% RSLogix 500 project Project 4.RSS, saved by version 8.30.00.16 %
PROJECT "UNTITLED"    % processor: Bul.1763 MicroLogix 1100 Series B %

PROGRAM FILES
  LAD 2 "MAIN"  5 rungs
  LAD 3 "IO"  8 rungs
  LAD 4 "CYCLE"  6 rungs
  LAD 5 "CONTROLS"  11 rungs

DATA FILES
  O0 OUTPUT  4 elements
  I1 INPUT  6 elements
  S2 STATUS  66 elements
  B3 BINARY  1 elements
  T4 TIMER  3 elements
  C5 COUNTER  1 elements
  R6 CONTROL  1 elements
  N7 INTEGER  3 elements
  F8 FLOAT  1 elements

LADDER 2 "MAIN"
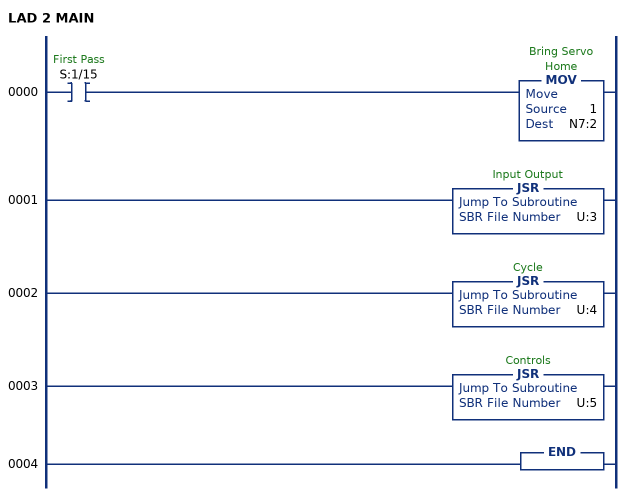
% Rung: 0 %
SOR XIC S:1/15 MOV 1 N7:2 EOR
%   S:1/15  "First Pass" %
%   N7:2  "Bring Servo Home" %
% Rung: 1 %
SOR JSR U:3 EOR
%   U:3  "Input Output" %
% Rung: 2 %
SOR JSR U:4 EOR
%   U:4  "Cycle" %
% Rung: 3 %
SOR JSR U:5 EOR
%   U:5  "Controls" %
% Rung: 4 %
SOR END EOR

LADDER 3 "IO"
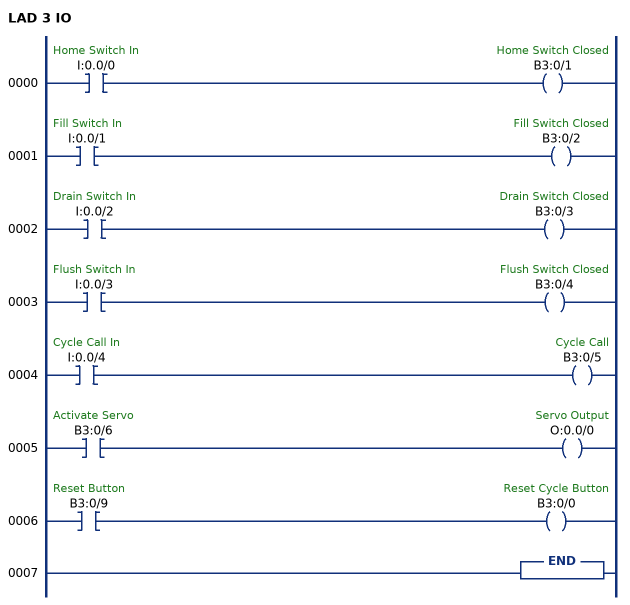
% Rung: 0 %
SOR XIC I:0.0/0 OTE B3:0/1 EOR
%   I:0.0/0  "Home Switch In" %
%   B3:0/1  "Home Switch Closed" %
% Rung: 1 %
SOR XIC I:0.0/1 OTE B3:0/2 EOR
%   I:0.0/1  "Fill Switch In" %
%   B3:0/2  "Fill Switch Closed" %
% Rung: 2 %
SOR XIC I:0.0/2 OTE B3:0/3 EOR
%   I:0.0/2  "Drain Switch In" %
%   B3:0/3  "Drain Switch Closed" %
% Rung: 3 %
SOR XIC I:0.0/3 OTE B3:0/4 EOR
%   I:0.0/3  "Flush Switch In" %
%   B3:0/4  "Flush Switch Closed" %
% Rung: 4 %
SOR XIC I:0.0/4 OTE B3:0/5 EOR
%   I:0.0/4  "Cycle Call In" %
%   B3:0/5  "Cycle Call" %
% Rung: 5 %
SOR XIC B3:0/6 OTE O:0.0/0 EOR
%   B3:0/6  "Activate Servo" %
%   O:0.0/0  "Servo Output" %
% Rung: 6 %
SOR XIC B3:0/9 OTE B3:0/0 EOR
%   B3:0/9  "Reset Button" %
%   B3:0/0  "Reset Cycle Button" %
% Rung: 7 %
SOR END EOR

LADDER 4 "CYCLE"
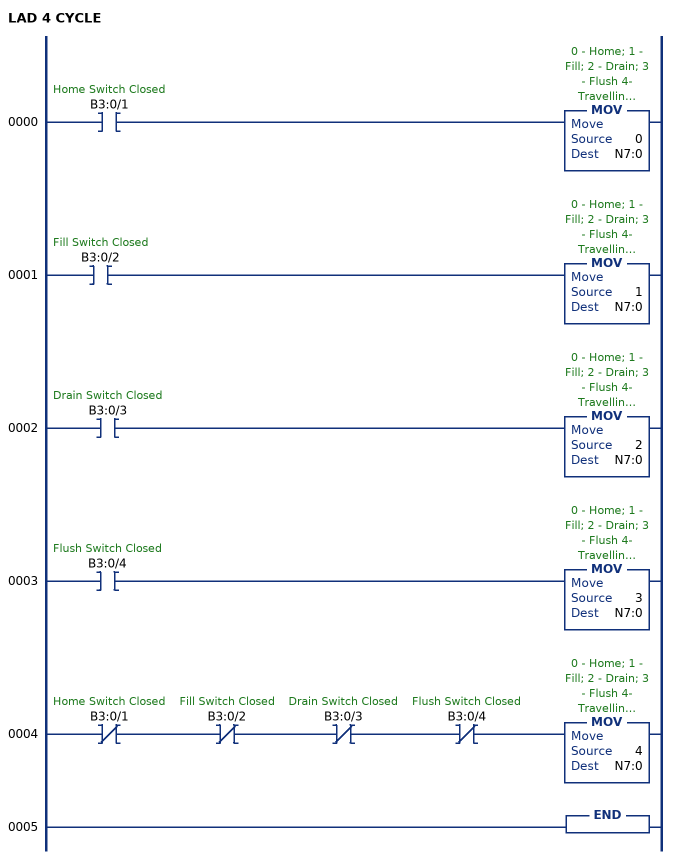
% Rung: 0 %
SOR XIC B3:0/1 MOV 0 N7:0 EOR
%   B3:0/1  "Home Switch Closed" %
%   N7:0  "0 - Home; 1 - Fill; 2 - Drain; 3 - Flush 4- Travelling Current Position" %
% Rung: 1 %
SOR XIC B3:0/2 MOV 1 N7:0 EOR
%   B3:0/2  "Fill Switch Closed" %
%   N7:0  "0 - Home; 1 - Fill; 2 - Drain; 3 - Flush 4- Travelling Current Position" %
% Rung: 2 %
SOR XIC B3:0/3 MOV 2 N7:0 EOR
%   B3:0/3  "Drain Switch Closed" %
%   N7:0  "0 - Home; 1 - Fill; 2 - Drain; 3 - Flush 4- Travelling Current Position" %
% Rung: 3 %
SOR XIC B3:0/4 MOV 3 N7:0 EOR
%   B3:0/4  "Flush Switch Closed" %
%   N7:0  "0 - Home; 1 - Fill; 2 - Drain; 3 - Flush 4- Travelling Current Position" %
% Rung: 4 %
SOR XIO B3:0/1 XIO B3:0/2 XIO B3:0/3 XIO B3:0/4 MOV 4 N7:0 EOR
%   B3:0/1  "Home Switch Closed" %
%   B3:0/2  "Fill Switch Closed" %
%   B3:0/3  "Drain Switch Closed" %
%   B3:0/4  "Flush Switch Closed" %
%   N7:0  "0 - Home; 1 - Fill; 2 - Drain; 3 - Flush 4- Travelling Current Position" %
% Rung: 5 %
SOR END EOR

LADDER 5 "CONTROLS"
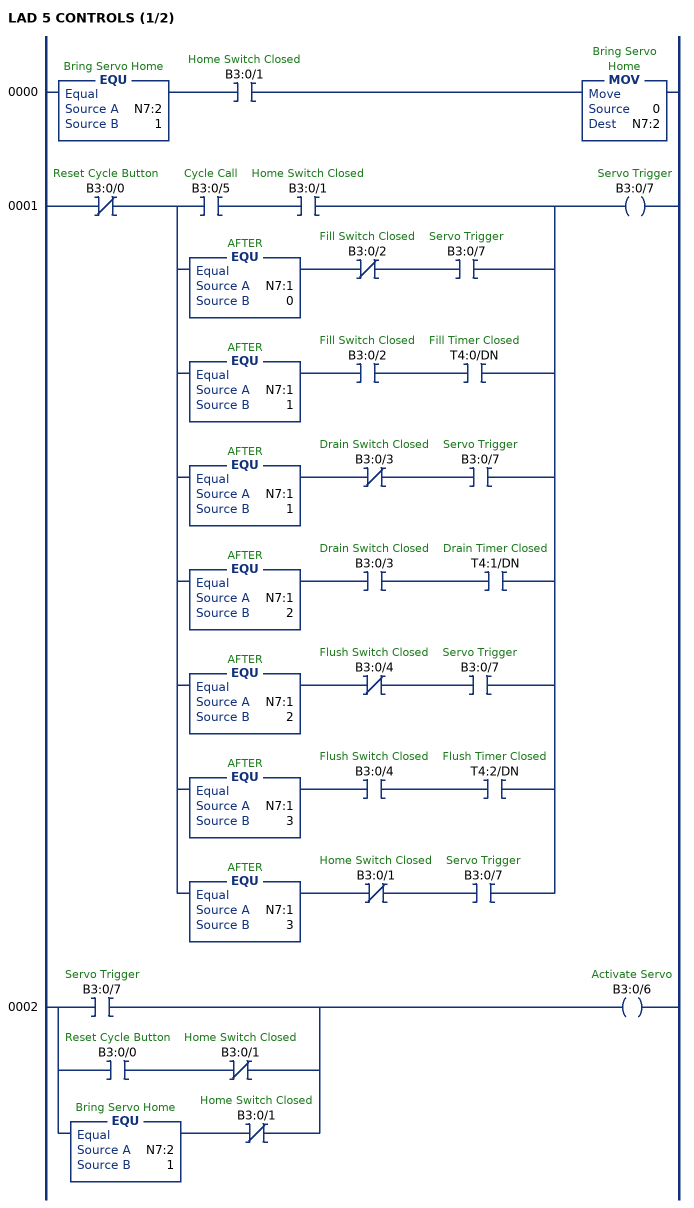
% Rung: 0 %
SOR EQU N7:2 1 XIC B3:0/1 MOV 0 N7:2 EOR
%   N7:2  "Bring Servo Home" %
%   B3:0/1  "Home Switch Closed" %
% Rung: 1 %
SOR XIO B3:0/0 BST XIC B3:0/5 XIC B3:0/1 NXB EQU N7:1 0 XIO B3:0/2 XIC B3:0/7 NXB EQU N7:1 1 XIC B3:0/2 XIC T4:0/DN NXB EQU N7:1 1 XIO B3:0/3 XIC B3:0/7 NXB EQU N7:1 2 XIC B3:0/3 XIC T4:1/DN NXB EQU N7:1 2 XIO B3:0/4 XIC B3:0/7 NXB EQU N7:1 3 XIC B3:0/4 XIC T4:2/DN NXB EQU N7:1 3 XIO B3:0/1 XIC B3:0/7 BND OTE B3:0/7 EOR
%   B3:0/0  "Reset Cycle Button" %
%   B3:0/5  "Cycle Call" %
%   B3:0/1  "Home Switch Closed" %
%   N7:1  AFTER %
%   B3:0/2  "Fill Switch Closed" %
%   B3:0/7  "Servo Trigger" %
%   T4:0/DN  "Fill Timer Closed" %
%   B3:0/3  "Drain Switch Closed" %
%   T4:1/DN  "Drain Timer Closed" %
%   B3:0/4  "Flush Switch Closed" %
%   T4:2/DN  "Flush Timer Closed" %
% Rung: 2 %
SOR BST XIC B3:0/7 NXB XIC B3:0/0 XIO B3:0/1 NXB EQU N7:2 1 XIO B3:0/1 BND OTE B3:0/6 EOR
%   B3:0/7  "Servo Trigger" %
%   B3:0/0  "Reset Cycle Button" %
%   B3:0/1  "Home Switch Closed" %
%   N7:2  "Bring Servo Home" %
%   B3:0/6  "Activate Servo" %

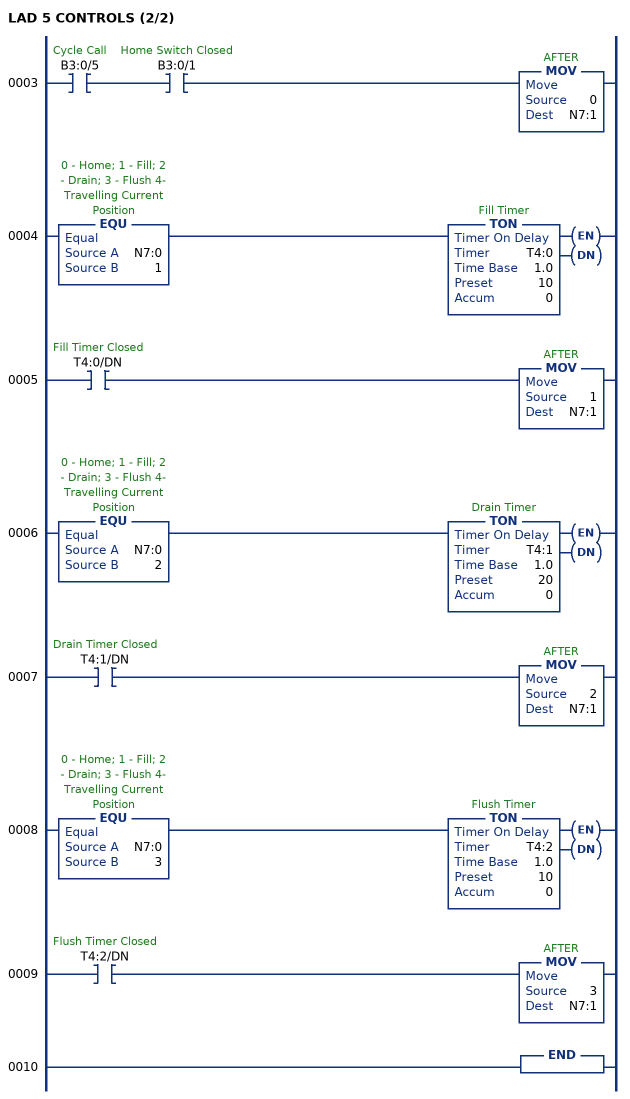
% Rung: 3 %
SOR XIC B3:0/5 XIC B3:0/1 MOV 0 N7:1 EOR
%   B3:0/5  "Cycle Call" %
%   B3:0/1  "Home Switch Closed" %
%   N7:1  AFTER %
% Rung: 4 %
SOR EQU N7:0 1 TON T4:0 1.0 10 0 EOR
%   N7:0  "0 - Home; 1 - Fill; 2 - Drain; 3 - Flush 4- Travelling Current Position" %
%   T4:0  "Fill Timer" %
% Rung: 5 %
SOR XIC T4:0/DN MOV 1 N7:1 EOR
%   T4:0/DN  "Fill Timer Closed" %
%   N7:1  AFTER %
% Rung: 6 %
SOR EQU N7:0 2 TON T4:1 1.0 20 0 EOR
%   N7:0  "0 - Home; 1 - Fill; 2 - Drain; 3 - Flush 4- Travelling Current Position" %
%   T4:1  "Drain Timer" %
% Rung: 7 %
SOR XIC T4:1/DN MOV 2 N7:1 EOR
%   T4:1/DN  "Drain Timer Closed" %
%   N7:1  AFTER %
% Rung: 8 %
SOR EQU N7:0 3 TON T4:2 1.0 10 0 EOR
%   N7:0  "0 - Home; 1 - Fill; 2 - Drain; 3 - Flush 4- Travelling Current Position" %
%   T4:2  "Flush Timer" %
% Rung: 9 %
SOR XIC T4:2/DN MOV 3 N7:1 EOR
%   T4:2/DN  "Flush Timer Closed" %
%   N7:1  AFTER %
% Rung: 10 %
SOR END EOR

OTHER DOCUMENTED ADDRESSES
  B3:0/8  "Take Servo Home"
  B3:0/10  "Fire Once"

DATA TABLE (non-zero values as saved)
DATA T4
% .PRE .ACC %
% T4:0 % 10 0
% T4:1 % 20 0
% T4:2 % 10 0
